// Machine control
TYPE ST_MachineControl:
STRUCT
    bReset: BIT;
    bStart: BIT;
    bStopNC: BIT;
    bManual: BIT;
    bAuto: BIT;
    bEmergStopNC: BIT;
END_STRUCT
END_TYPE

(* stored: Version 1.1.0.1
   DUT ST_MachineControl: Id {b772704c-c125-48f7-a7ed-223f738cbb87} *)
